// TIA Portal V17 export
// export: Created 2025-03-07T09:18:19.1138897Z, ExportSetting WithDefaults, DisplayName Totally Integrated Automation Portal, DisplayVersion V17 Update 8, DisplayName TIA Portal Openness, DisplayVersion V17 Update 8, DisplayName TIA Portal Version Control Interface, DisplayVersion V17, DisplayName SINAMICS Startdrive Advanced, DisplayVersion V17 SP2, DisplayName SINAMICS Startdrive G110M, G120, G120C, G120D, G120P, G115D, DisplayVersion V17 SP2, DisplayName SINAMICS Startdrive G130, G150, S120, S150, SINAMICS MV, S210, DisplayVersion V17 SP2, DisplayName STEP 7 Professional, DisplayVersion V17 Update 8, DisplayName SINUMERIK ONE STEP 7 Toolbox, DisplayVersion V17 Update 12, DisplayName SINUMERIK 840D sl STEP 7 Toolbox, DisplayVersion V17 Update 12, DisplayName STEP 7 Safety, DisplayVersion V17 Update 6, DisplayName WinCC Advanced, DisplayVersion V17 Update 8
DATA_BLOCK "DB1421_PROGRESSIVE_LUBRICATION_WITH_GREASE"   // DB1421
AUTHOR : ETXETAR
VERSION : 1.0
// stored: AutoNumber false, DBAccessibleFromOPCUA true, DBAccessibleFromWebserver true, InstanceOfName FB1403_PROGRESSIVE_LUBRICATION_WITH_GREASE, InstanceOfType FB
"FB1403_PROGRESSIVE_LUBRICATION_WITH_GREASE"
   // VAR_INPUT
   //    OPTIONS_0 : Byte;
   //    OPTIONS_1 : Byte;
   //    TIME_VALVE_1 : Time;
   //    TIME_VALVE_2 : Time;
   //    TIME_VALVE_3 : Time;
   //    TIME_VALVE_4 : Time;
   //    PULSES_PER_CYCLE_VALVE_1 : Int;
   //    PULSES_PER_CYCLE_VALVE_2 : Int;
   //    PULSES_PER_CYCLE_VALVE_3 : Int;
   //    PULSES_PER_CYCLE_VALVE_4 : Int;
   //    BREAKER : Bool;
   //    LOW_LEVEL_ALM : Bool;
   //    OVERPRESSURE_ALM : Bool;
   //    LUBRICATION_DONE_1 : Bool;
   //    LUBRICATION_DONE_2 : Bool;
   //    LUBRICATION_DONE_3 : Bool;
   //    LUBRICATION_DONE_4 : Bool;
   //    LUBRICATION_DONE_5 : Bool;
   //    LUBRICATION_DONE_6 : Bool;
   //    LUBRICATION_DONE_7 : Bool;
   //    LUBRICATION_DONE_8 : Bool;
   //    LUBRICATION_DONE_9 : Bool;
   //    SWITCH_ON_VALVE_1_DIST_REQ_AXIS_1 : Bool;
   //    SWITCH_ON_VALVE_1_DIST_REQ_AXIS_2 : Bool;
   //    SWITCH_ON_VALVE_2_DIST_REQ_AXIS_1 : Bool;
   //    SWITCH_ON_VALVE_2_DIST_REQ_AXIS_2 : Bool;
   //    SWITCH_ON_VALVE_3_DIST_REQ : Bool;
   //    SWITCH_ON_VALVE_4_DIST_REQ : Bool;
   //    HMI_REQ_LINE_VALVE_1 : Bool;
   //    HMI_REQ_LINE_VALVE_2 : Bool;
   //    HMI_REQ_LINE_VALVE_3 : Bool;
   //    HMI_REQ_LINE_VALVE_4 : Bool;
   // END_VAR
   // VAR_OUTPUT
   //    HMI_POWER_UP_COND_OFF_VALVE_1 : Bool;
   //    HMI_POWER_UP_COND_ON_VALVE_1 : Bool;
   //    HMI_POWER_UP_EXECU_LEFT_VALVE_1 : Bool;
   //    HMI_POWER_UP_EXECU_RIGHT_VALVE_1 : Bool;
   //    HMI_POWER_UP_COND_OFF_VALVE_2 : Bool;
   //    HMI_POWER_UP_COND_ON_VALVE_2 : Bool;
   //    HMI_POWER_UP_EXECU_LEFT_VALVE_2 : Bool;
   //    HMI_POWER_UP_EXECU_RIGHT_VALVE_2 : Bool;
   //    HMI_POWER_UP_COND_OFF_VALVE_3 : Bool;
   //    HMI_POWER_UP_COND_ON_VALVE_3 : Bool;
   //    HMI_POWER_UP_EXECU_LEFT_VALVE_3 : Bool;
   //    HMI_POWER_UP_EXECU_RIGHT_VALVE_3 : Bool;
   //    HMI_POWER_UP_COND_OFF_VALVE_4 : Bool;
   //    HMI_POWER_UP_COND_ON_VALVE_4 : Bool;
   //    HMI_POWER_UP_EXECU_LEFT_VALVE_4 : Bool;
   //    HMI_POWER_UP_EXECU_RIGHT_VALVE_4 : Bool;
   //    MOTOR : Bool;
   //    VALVE_1 : Bool;
   //    VALVE_2 : Bool;
   //    VALVE_3 : Bool;
   //    VALVE_4 : Bool;
   // END_VAR
   // VAR RETAIN
   //    BREAKER_ALARM : Bool;
   //    LOW_LEVEL_ALARM : Bool;
   //    OVERPRESSURE_ALARM : Bool;
   //    LUBRICATION_DONE_1_ALARM : Bool;
   //    LUBRICATION_DONE_2_ALARM : Bool;
   //    LUBRICATION_DONE_3_ALARM : Bool;
   //    LUBRICATION_DONE_4_ALARM : Bool;
   //    DATA_VALVE_1 : Struct
   //       SWITCH_ON_GENERAL_CONDITIONS : Bool;
   //       SWITCH_ON_INITIAL_CONDITIONS : Bool;
   //       SWITCH_ON_MANUAL_REQUEST : Bool;
   //       SWITCH_ON_AUTO_REQUEST : Bool;
   //       SWITCH_ON_TIME_REQUEST : Bool;
   //       SWITCH_ON_GLOBAL_REQUEST : Bool;
   //       SWITCH_ON_CMM : Bool;
   //       SWITCH_ON : Bool;
   //       IN_SERVICE : Bool;
   //       SWITCH_OFF_GENERAL_CONDITIONS : Bool;
   //       SWITCH_OFF_INITIAL_CONDITIONS : Bool;
   //       SWITCH_OFF_MANUAL_REQUEST : Bool;
   //       SWITCH_OFF_AUTO_REQUEST : Bool;
   //       SWITCH_OFF_GLOBAL_REQUEST : Bool;
   //       SWITCH_OFF_CMM : Bool;
   //       SWITCH_OFF : Bool;
   //       OUT_OF_SERVICE : Bool;
   //       TIMER_1 : TON_TIME;
   //       PULSE_1 : Bool;
   //       PULSE_2 : Bool;
   //    END_STRUCT;
   //    DATA_VALVE_2 : Struct
   //       SWITCH_ON_GENERAL_CONDITIONS : Bool;
   //       SWITCH_ON_INITIAL_CONDITIONS : Bool;
   //       SWITCH_ON_MANUAL_REQUEST : Bool;
   //       SWITCH_ON_AUTO_REQUEST : Bool;
   //       SWITCH_ON_TIME_REQUEST : Bool;
   //       SWITCH_ON_GLOBAL_REQUEST : Bool;
   //       SWITCH_ON_CMM : Bool;
   //       SWITCH_ON : Bool;
   //       IN_SERVICE : Bool;
   //       SWITCH_OFF_GENERAL_CONDITIONS : Bool;
   //       SWITCH_OFF_INITIAL_CONDITIONS : Bool;
   //       SWITCH_OFF_MANUAL_REQUEST : Bool;
   //       SWITCH_OFF_AUTO_REQUEST : Bool;
   //       SWITCH_OFF_GLOBAL_REQUEST : Bool;
   //       SWITCH_OFF_CMM : Bool;
   //       SWITCH_OFF : Bool;
   //       OUT_OF_SERVICE : Bool;
   //       TIMER_1 : TON_TIME;
   //       PULSE_1 : Bool;
   //       PULSE_2 : Bool;
   //    END_STRUCT;
   //    DATA_VALVE_3 : Struct
   //       SWITCH_ON_GENERAL_CONDITIONS : Bool;
   //       SWITCH_ON_INITIAL_CONDITIONS : Bool;
   //       SWITCH_ON_MANUAL_REQUEST : Bool;
   //       SWITCH_ON_AUTO_REQUEST : Bool;
   //       SWITCH_ON_TIME_REQUEST : Bool;
   //       SWITCH_ON_GLOBAL_REQUEST : Bool;
   //       SWITCH_ON_CMM : Bool;
   //       SWITCH_ON : Bool;
   //       IN_SERVICE : Bool;
   //       SWITCH_OFF_GENERAL_CONDITIONS : Bool;
   //       SWITCH_OFF_INITIAL_CONDITIONS : Bool;
   //       SWITCH_OFF_MANUAL_REQUEST : Bool;
   //       SWITCH_OFF_AUTO_REQUEST : Bool;
   //       SWITCH_OFF_GLOBAL_REQUEST : Bool;
   //       SWITCH_OFF_CMM : Bool;
   //       SWITCH_OFF : Bool;
   //       OUT_OF_SERVICE : Bool;
   //       TIMER_1 : TON_TIME;
   //       PULSE_1 : Bool;
   //       PULSE_2 : Bool;
   //    END_STRUCT;
   //    DATA_VALVE_4 : Struct
   //       SWITCH_ON_GENERAL_CONDITIONS : Bool;
   //       SWITCH_ON_INITIAL_CONDITIONS : Bool;
   //       SWITCH_ON_MANUAL_REQUEST : Bool;
   //       SWITCH_ON_AUTO_REQUEST : Bool;
   //       SWITCH_ON_TIME_REQUEST : Bool;
   //       SWITCH_ON_GLOBAL_REQUEST : Bool;
   //       SWITCH_ON_CMM : Bool;
   //       SWITCH_ON : Bool;
   //       IN_SERVICE : Bool;
   //       SWITCH_OFF_GENERAL_CONDITIONS : Bool;
   //       SWITCH_OFF_INITIAL_CONDITIONS : Bool;
   //       SWITCH_OFF_MANUAL_REQUEST : Bool;
   //       SWITCH_OFF_AUTO_REQUEST : Bool;
   //       SWITCH_OFF_GLOBAL_REQUEST : Bool;
   //       SWITCH_OFF_CMM : Bool;
   //       SWITCH_OFF : Bool;
   //       OUT_OF_SERVICE : Bool;
   //       TIMER_1 : TON_TIME;
   //       PULSE_1 : Bool;
   //       PULSE_2 : Bool;
   //    END_STRUCT;
   //    CYCLE_IN_PROCESS : Bool;
   //    ALL_LUBRICATION_DONE : Bool;
   //    ALL_LUBRICATION_DONE_DELAYED : Bool;
   //    SWITCH_ON_MOTOR_REQUEST : Bool;
   //    ANY_CYCLE_NOT_DONE : Bool;
   //    CYCLE_FINISHED_1 : Bool;
   //    CYCLE_FINISHED_2 : Bool;
   //    CYCLE_FINISHED_3 : Bool;
   //    CYCLE_FINISHED_4 : Bool;
   //    MANUAL_REQUEST_HELP : Bool;
   //    SWITCH_ON_GENERAL_CONDITION_HELP : Bool;
   //    SWITCH_ON_INITIAL_CONDITION_HELP : Bool;
   //    SWITCH_OFF_GENERAL_CONDITION_HELP : Bool;
   //    SWITCH_OFF_INITIAL_CONDITION_HELP : Bool;
   //    ANY_ACTIVE_ALARM : Bool;
   //    SEOC_ALARMS : Bool;
   //    WARNINGS : Bool;
   //    WARNINGS_GONE : Bool;
   //    TIMER_AUX_SWTICH_ON_MOTOR : TON_TIME;
   //    TIMER_ALL_LUBRICATION_DONE : TON_TIME;
   //    TIMER_LOW_LEVEL_ALM : TON_TIME;
   //    TIMER_OVERPRESSURE_ALM : TON_TIME;
   //    TIMER_ANY_CYCLE_NOT_DONE : TON_TIME;
   //    TIMER_RUN_NIGHT_TEST : TON_TIME;
   //    COUNTER_1 { S7_SetPoint := 'True'} : CTU_INT;
   //    COUNTER_2 { S7_SetPoint := 'True'} : CTU_INT;
   //    COUNTER_3 { S7_SetPoint := 'True'} : CTU_INT;
   //    COUNTER_4 { S7_SetPoint := 'True'} : CTU_INT;
   //    SEQ_GLOBAL_AUTO_REQ : Bool;
   //    PULSE_1 : Bool;
   //    PULSE_2 : Bool;
   //    PULSE_3 : Bool;
   //    PULSE_4 : Bool;
   //    PULSE_5 : Bool;
   //    PULSE_6 : Bool;
   //    PULSE_7 : Bool;
   //    PULSE_8 : Bool;
   //    VALVE_1_AXIS_1_DIST_MEM_REQ : Bool;
   //    VALVE_1_AXIS_2_DIST_MEM_REQ : Bool;
   //    VALVE_2_AXIS_1_DIST_MEM_REQ : Bool;
   //    VALVE_2_AXIS_2_DIST_MEM_REQ : Bool;
   //    VALVE_1_AXIS_1_2_DIST_REQ : Bool;
   //    VALVE_2_AXIS_1_2_DIST_REQ : Bool;
   // END_VAR
BEGIN
END_DATA_BLOCK
